(* PLC project BlogProject.project, CODESYS CODESYS V3.5 SP14 Patch 3 *)
(* stored: creationDateTime 2021-10-07T21:08:10.6540194, modificationDateTime 2021-10-07T20:40:20.1109198 *)

PROGRAM FSM_Kernel
  VAR
    Core : MC_CORE;
  END_VAR

            Core(System:=ADR(System1));
          
END_PROGRAM
